{attribute addProperty BoxType "AT2025-0250-0020"}
{attribute addProperty Id "A_0074_AT2000_5250_0017_AT2000_5250AT2000_3DCFC8D064080"}
{attribute addProperty CRC "3573915941"}
{attribute addProperty SizeInBites "640"}
{attribute addProperty SizeInBytes "80"}
TYPE A_0062_AT2025_0250_0020_AT2025_0250_D505A125 EXTENDS AT2025_9506A482 :
STRUCT
	{attribute addProperty Name "A_0074_AT2000_5250_0017_AT2000_5250"}
	A_0074_AT2000_5250_0017_AT2000_5250 : AT2000_3DCFC8D0;
END_STRUCT
END_TYPE

(* stored: Version 1.2.0.0, ProductVersion 3.1.4024.9
   DUT A_0062_AT2025_0250_0020_AT2025_0250_D505A125: Id {762f0245-ea43-4ffb-85cc-f55fb4226d4b} *)
